INTERFACE I_ComponentBase EXTENDS I_Base

METHOD AllowHMIControl
VAR_INPUT
END_VAR
END_METHOD

METHOD BlockHMIControl 
VAR_INPUT
END_VAR
END_METHOD

PROPERTY CurrentAlarmSeverity : TcEventSeverity
GET
END_GET
END_PROPERTY

PROPERTY InSimulation : Bool
GET
END_GET
SET
END_SET
END_PROPERTY

PROPERTY Name : String
GET
END_GET
SET
END_SET
END_PROPERTY

METHOD Reset
VAR_INPUT
END_VAR
END_METHOD

END_INTERFACE

(* stored: Version 1.1.0.1, ProductVersion 3.1.4024.14
   Itf I_ComponentBase: Id {9e5694a3-27f3-4799-8b1e-d3da44d6be86}
   Folder Methods: Id {1e2e9b13-8035-499a-b994-72999b980d9e}
   Folder Properties: Id {253b39ea-054f-4168-a4fb-b621c19f84e8}
   Method AllowHMIControl: Id {0dc61043-a0c4-48c3-bf79-c3b3d185c81e}
   Method BlockHMIControl: Id {13beeb00-1a58-495c-8e9e-479a85cd7211}
   Property CurrentAlarmSeverity: Id {77d85cd6-9dc8-40a3-b94b-a66fee89834f}
   Get Get: Id {ab95067c-f7b0-450d-b5e2-ab7c12ff6232}
   Property InSimulation: Id {2f6a6102-2fd3-43af-871c-13ac4383092a}
   Get Get: Id {a77f9960-2ef4-4fcd-a23f-8767b1ac8142}
   Set Set: Id {0a6c4719-2d36-4a6a-bbb0-b0b5ea45e1d1}
   Property Name: Id {a26bdb86-fe9d-474f-bcaa-1df8613d0cb8}
   Get Get: Id {77076a69-c81d-42cb-9044-99e46338a24c}
   Set Set: Id {aff21efc-e535-4d77-8755-f342ed6752a4}
   Method Reset: Id {30edff56-7568-45fa-b6e7-07d6ee74dcf3} *)
